{attribute addProperty BoxType "EJ2521-0224-0016"}
{attribute addProperty Id "Sel_Ack_End_counterBIT10.1251Ramp_activeBIT10.1252ErrorBIT10.1257Sync_errorBIT10.12514TxPDO_ToggleBIT10.12516"}
{attribute addProperty CRC "813189523"}
{attribute addProperty SizeInBites "16"}
{attribute addProperty SizeInBytes "2"}
TYPE Status_30784993 :
STRUCT
	{attribute addProperty Name "Sel_Ack_End_counter"}
	Sel_Ack_End_counter : BIT;
	{attribute addProperty Name "Ramp_active"}
	Ramp_active : BIT;
	{attribute 'hide'}
	reserve_1_BIT_0 : BIT;
	{attribute 'hide'}
	reserve_1_BIT_1 : BIT;
	{attribute 'hide'}
	reserve_1_BIT_2 : BIT;
	{attribute 'hide'}
	reserve_1_BIT_3 : BIT;
	{attribute addProperty Name "Error"}
	Error : BIT;
	{attribute 'hide'}
	reserve_2_BIT_0 : BIT;
	{attribute 'hide'}
	reserve_2_BIT_1 : BIT;
	{attribute 'hide'}
	reserve_2_BIT_2 : BIT;
	{attribute 'hide'}
	reserve_2_BIT_3 : BIT;
	{attribute 'hide'}
	reserve_2_BIT_4 : BIT;
	{attribute 'hide'}
	reserve_2_BIT_5 : BIT;
	{attribute addProperty Name "Sync_error"}
	Sync_error : BIT;
	{attribute 'hide'}
	reserve_3 : BIT;
	{attribute addProperty Name "TxPDO_Toggle"}
	TxPDO_Toggle : BIT;
END_STRUCT
END_TYPE

(* stored: Version 1.2.0.0, ProductVersion 3.1.4024.9
   DUT Status_30784993: Id {eeb6d667-8778-4662-904c-cb0cdaae8203} *)
